FUNCTION_BLOCK FB_EventBuffer
VAR
	fbMemRingBuffer : FB_MemRingBuffer;
	BufferArray  : ARRAY[0..NUMBER_BYTES_FOR_ST_EVENT] OF BYTE; (* Buffer memory used by FB_MemRingBuffer function block *)
END_VAR

VAR CONSTANT
	ST_EVENT_SiZE : UDINT := SIZEOF(ST_Event); // size of a type
	MAX_NUMBER_ST_EVENT : UDINT := 5;
	NUMBER_BYTES_FOR_ST_EVENT : UDINT := MAX_NUMBER_ST_EVENT * ST_EVENT_SiZE;
END_VAR

METHOD PUBLIC AddEvent
VAR_INPUT
	stEvent : REFERENCE TO ST_Event;
END_VAR
VAR_OUTPUT
	bError : BOOL;
END_VAR
fbMemRingBuffer.A_AddTail(pWrite := ADR(stEvent),
							cbWrite := SIZEOF(stEvent),
							pBuffer := ADR(BufferArray),
							cbBuffer := SIZEOF(BufferArray));

bError := NOT fbMemRingBuffer.bOk;
END_METHOD

METHOD GetRemoveEvent
VAR_OUTPUT
	stEvent : ST_Event;
	bError : BOOL;
END_VAR
fbMemRingBuffer.A_RemoveHead(pRead := ADR(stEvent),
							cbRead := SIZEOF(stEvent),
							pBuffer := ADR(BufferArray),
							cbBuffer := SIZEOF(BufferArray));
							
bError := NOT fbMemRingBuffer.bOk;
END_METHOD

END_FUNCTION_BLOCK

(* stored: Version 1.1.0.1, ProductVersion 3.1.4024.12
   POU FB_EventBuffer: Id {49471cf7-86f2-4e1c-82b4-7d84c2c029c9}, SpecialFunc None
   Method AddEvent: Id {ee1470b7-ac79-4855-82f0-5b235754a129}
   Method GetRemoveEvent: Id {bd20d893-0e15-44ab-a492-2fa710bb5162} *)
